PROGRAM PRG_PAOL_03_LightboxSeparatorCtrl
VAR

	rtrigDriveFaultAcknowledge		: R_TRIG;
	tofDriveFaultAcknowledge			: TOF;

	tonSeparationDriveDelayStart		: TON;
END_VAR
VAR // added by the converter: edge detectors and wires of the graphical bodies
    _w1, _w2 : BOOL;
END_VAR

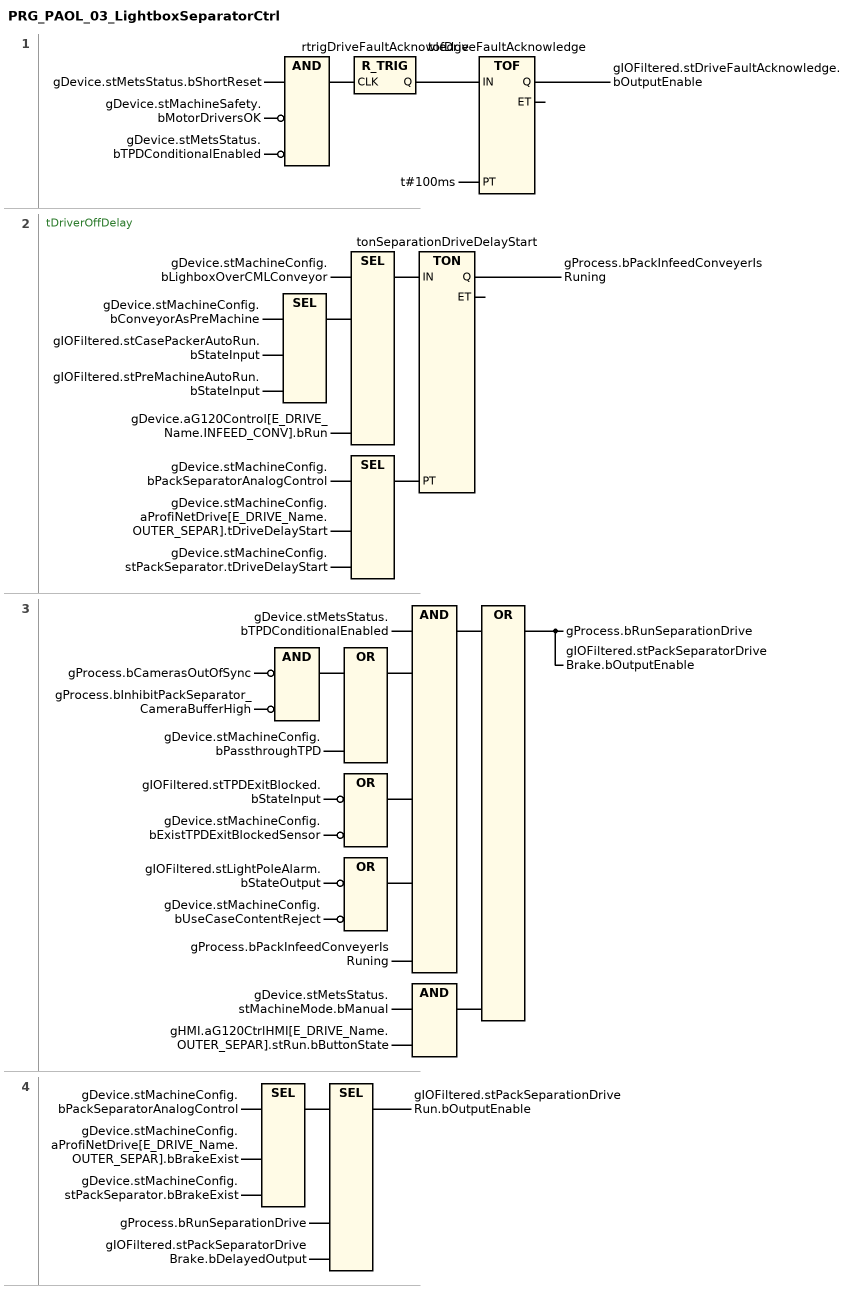
// NETWORK 1
rtrigDriveFaultAcknowledge(CLK := gDevice.stMetsStatus.bShortReset AND NOT gDevice.stMachineSafety.bMotorDriversOK AND NOT gDevice.stMetsStatus.bTPDConditionalEnabled); // R_TRIG
tofDriveFaultAcknowledge(IN := rtrigDriveFaultAcknowledge.Q, PT := t#100ms); // TOF
gIOFiltered.stDriveFaultAcknowledge.bOutputEnable := tofDriveFaultAcknowledge.Q;

// NETWORK 2
// tDriverOffDelay
tonSeparationDriveDelayStart(IN := SEL(gDevice.stMachineConfig.bLighboxOverCMLConveyor, SEL(gDevice.stMachineConfig.bConveyorAsPreMachine, gIOFiltered.stCasePackerAutoRun.bStateInput, gIOFiltered.stPreMachineAutoRun.bStateInput), gDevice.aG120Control[E_DRIVE_Name.INFEED_CONV].bRun), PT := SEL(gDevice.stMachineConfig.bPackSeparatorAnalogControl, gDevice.stMachineConfig.aProfiNetDrive[E_DRIVE_Name.OUTER_SEPAR].tDriveDelayStart, gDevice.stMachineConfig.stPackSeparator.tDriveDelayStart)); // TON
gProcess.bPackInfeedConveyerIsRuning := tonSeparationDriveDelayStart.Q;

// NETWORK 3
_w1 := gDevice.stMetsStatus.bTPDConditionalEnabled AND (NOT gProcess.bCamerasOutOfSync AND NOT gProcess.bInhibitPackSeparator_CameraBufferHigh OR gDevice.stMachineConfig.bPassthroughTPD) AND (NOT gIOFiltered.stTPDExitBlocked.bStateInput OR NOT gDevice.stMachineConfig.bExistTPDExitBlockedSensor) AND (NOT gIOFiltered.stLightPoleAlarm.bStateOutput OR NOT gDevice.stMachineConfig.bUseCaseContentReject) AND gProcess.bPackInfeedConveyerIsRuning OR gDevice.stMetsStatus.stMachineMode.bManual AND gHMI.aG120CtrlHMI[E_DRIVE_Name.OUTER_SEPAR].stRun.bButtonState;
gProcess.bRunSeparationDrive := _w1;
gIOFiltered.stPackSeparatorDriveBrake.bOutputEnable := _w1;

// NETWORK 4
gIOFiltered.stPackSeparationDriveRun.bOutputEnable := SEL(SEL(gDevice.stMachineConfig.bPackSeparatorAnalogControl, gDevice.stMachineConfig.aProfiNetDrive[E_DRIVE_Name.OUTER_SEPAR].bBrakeExist, gDevice.stMachineConfig.stPackSeparator.bBrakeExist), gProcess.bRunSeparationDrive, gIOFiltered.stPackSeparatorDriveBrake.bDelayedOutput);

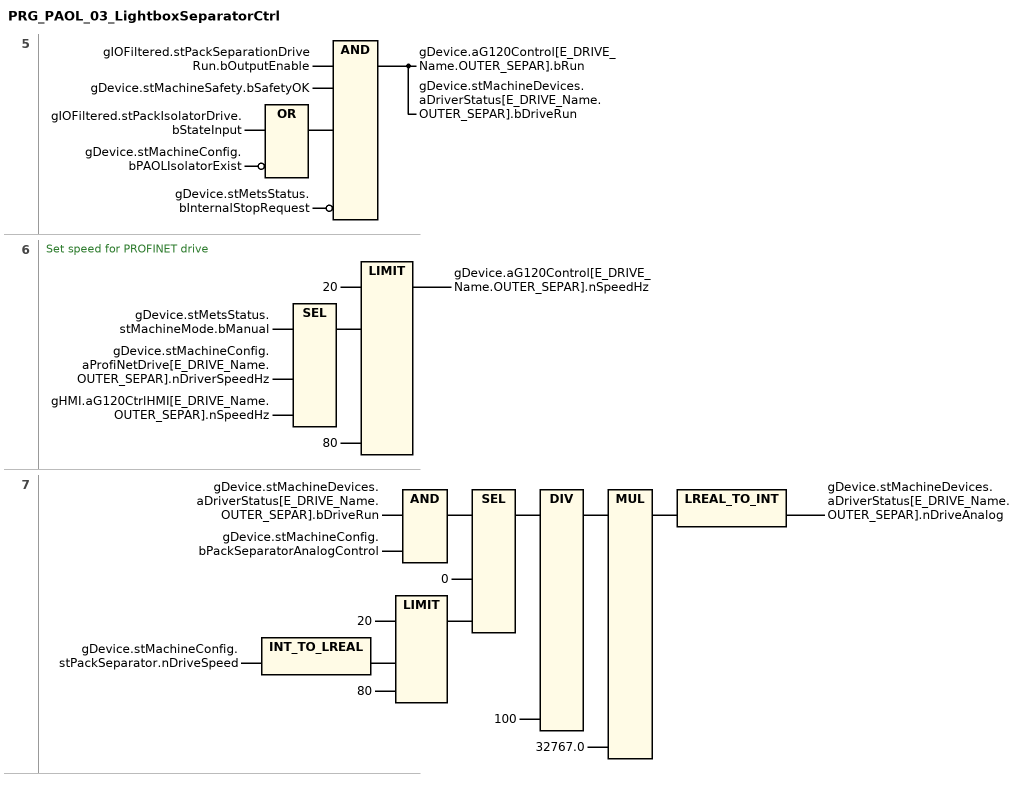
// NETWORK 5
_w2 := gIOFiltered.stPackSeparationDriveRun.bOutputEnable AND gDevice.stMachineSafety.bSafetyOK AND (gIOFiltered.stPackIsolatorDrive.bStateInput OR NOT gDevice.stMachineConfig.bPAOLIsolatorExist) AND NOT gDevice.stMetsStatus.bInternalStopRequest;
gDevice.aG120Control[E_DRIVE_Name.OUTER_SEPAR].bRun := _w2;
gDevice.stMachineDevices.aDriverStatus[E_DRIVE_Name.OUTER_SEPAR].bDriveRun := _w2;

// NETWORK 6
// Set speed for PROFINET drive
gDevice.aG120Control[E_DRIVE_Name.OUTER_SEPAR].nSpeedHz := LIMIT(20, SEL(gDevice.stMetsStatus.stMachineMode.bManual, gDevice.stMachineConfig.aProfiNetDrive[E_DRIVE_Name.OUTER_SEPAR].nDriverSpeedHz, gHMI.aG120CtrlHMI[E_DRIVE_Name.OUTER_SEPAR].nSpeedHz), 80);

// NETWORK 7
gDevice.stMachineDevices.aDriverStatus[E_DRIVE_Name.OUTER_SEPAR].nDriveAnalog := LREAL_TO_INT((SEL(gDevice.stMachineDevices.aDriverStatus[E_DRIVE_Name.OUTER_SEPAR].bDriveRun AND gDevice.stMachineConfig.bPackSeparatorAnalogControl, 0, LIMIT(20, INT_TO_LREAL(gDevice.stMachineConfig.stPackSeparator.nDriveSpeed), 80)) / 100) * 32767.0);

END_PROGRAM

(* stored: Version 1.1.0.1
   POU PRG_PAOL_03_LightboxSeparatorCtrl: Id {8659c6e2-bf38-4c3a-821b-19b3e9c2fe97}, SpecialFunc None *)
